FUNCTION_BLOCK GR_plant_Without_NDT
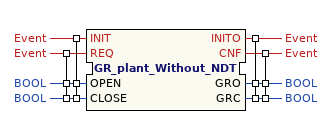
  EVENT_INPUT
    INIT WITH OPEN, CLOSE;
    REQ WITH OPEN, CLOSE;
  END_EVENT
  EVENT_OUTPUT
    INITO WITH GRO, GRC;
    CNF WITH GRO, GRC;
  END_EVENT
  VAR_INPUT
    OPEN : BOOL;
    CLOSE : BOOL;
  END_VAR
  VAR_OUTPUT
    GRO : BOOL;
    GRC : BOOL;
  END_VAR
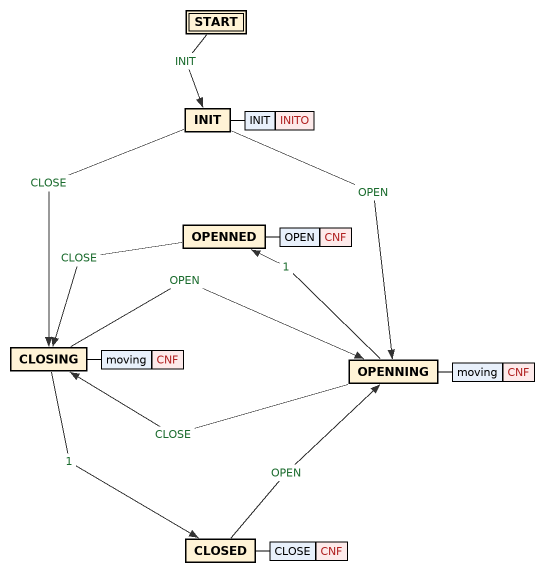
  EC_STATES
    START;
    INIT : INIT -> INITO;
    OPENNED : OPEN -> CNF;
    CLOSED : CLOSE -> CNF;
    OPENNING : moving -> CNF;
    CLOSING : moving -> CNF;
  END_STATES
  EC_TRANSITIONS
    CLOSING TO CLOSED := 1;
    CLOSED TO OPENNING := OPEN;
    OPENNING TO OPENNED := 1;
    OPENNED TO CLOSING := CLOSE;
    START TO INIT := INIT;
    CLOSING TO OPENNING := OPEN;
    OPENNING TO CLOSING := CLOSE;
    INIT TO CLOSING := CLOSE;
    INIT TO OPENNING := OPEN;
  END_TRANSITIONS
  ALGORITHM INIT IN ST:
GRO := FALSE;
GRC := FALSE;
  END_ALGORITHM
  ALGORITHM OPEN IN ST:
GRO := TRUE;
GRC := FALSE;
  END_ALGORITHM
  ALGORITHM moving IN ST:
GRO := FALSE;
GRC := FALSE;
  END_ALGORITHM
  ALGORITHM CLOSE IN ST:
GRC := TRUE;
GRO := FALSE;
  END_ALGORITHM
  ALGORITHM STOP IN ST:
GRO := FALSE;
GRC := FALSE;
  END_ALGORITHM
END_FUNCTION_BLOCK
